// TIA Portal project "Conveyor_LAD_V16_20260903" (V16)

(* hardware
DEVICE "S7-1200 station_1"  S7-1200 Station
   slot 0: "Rack_0"  S7-1200 Rack  Rack  V1.0
   slot 1: "PLC_Conveyor"  CPU 1214C DC/DC/DC  6ES7 214-1AG40-0XB0  V4.4
*)

// ===== PLC "PLC_Conveyor"  CPU 1214C DC/DC/DC =====

VAR_GLOBAL   // PLC tag table "Conveyor_IO_LAD"
   "Conveyor_StartButton" AT %I0.0 : Bool;
   "Conveyor_StopOK" AT %I0.1 : Bool;
   "Conveyor_EStopOK" AT %I0.2 : Bool;
   "Conveyor_OverloadOK" AT %I0.3 : Bool;
   "Conveyor_JamSensor" AT %I0.4 : Bool;
   "Conveyor_ResetButton" AT %I0.5 : Bool;
   "Conveyor_MotorCmd" AT %Q0.0 : Bool;
   "Conveyor_RunLamp" AT %Q0.1 : Bool;
   "Conveyor_FaultLamp" AT %Q0.2 : Bool;
END_VAR

DATA_BLOCK "DB_Conveyor_LAD"   // DB2
{ S7_Optimized_Access := 'TRUE' }
VERSION : 0.1
// stored: InstanceOfName FB_Conveyor_LAD
"FB_Conveyor_LAD"
BEGIN
END_DATA_BLOCK

FUNCTION_BLOCK "FB_Conveyor_LAD"   // FB2, LAD
{ S7_Optimized_Access := 'TRUE' }
   VAR_INPUT
      FirstScan : Bool;
      StartButton : Bool;
      StopOK : Bool;
      EStopOK : Bool;
      OverloadOK : Bool;
      JamSensor : Bool;
      ResetButton : Bool;
      JamTime : Time := T#5s;
   END_VAR
   VAR_OUTPUT
      MotorCmd : Bool;
      RunLamp : Bool;
      FaultLamp : Bool;
   END_VAR
   VAR
      StartPrev : Bool := FALSE;
      RunLatch : Bool := FALSE;
      FaultLatch : Bool := FALSE;
      JamTimer : TON_TIME;
   END_VAR
BEGIN

REGION Network 1: 01 - First scan: reset run latch
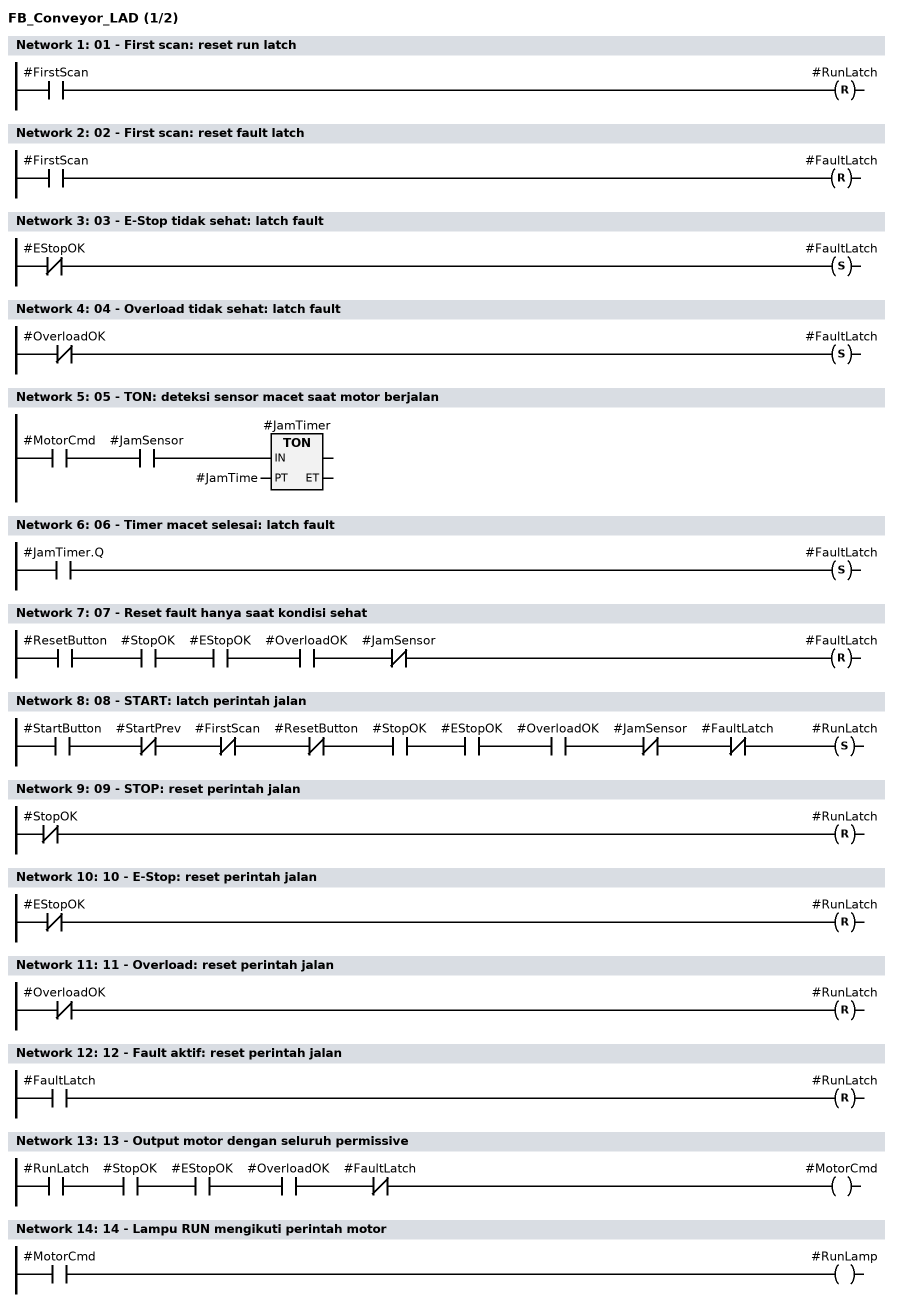
   RUNG wire#powerrail
      Contact( #FirstScan )
      R_Coil( #RunLatch )
   END_RUNG
   // the same network as SCL:
   IF #FirstScan THEN #RunLatch := FALSE; END_IF;
END_REGION

REGION Network 2: 02 - First scan: reset fault latch
   RUNG wire#powerrail
      Contact( #FirstScan )
      R_Coil( #FaultLatch )
   END_RUNG
   // the same network as SCL:
   IF #FirstScan THEN #FaultLatch := FALSE; END_IF;
END_REGION

REGION Network 3: 03 - E-Stop tidak sehat: latch fault
   RUNG wire#powerrail
      I_Contact( #EStopOK )
      S_Coil( #FaultLatch )
   END_RUNG
   // the same network as SCL:
   IF NOT #EStopOK THEN #FaultLatch := TRUE; END_IF;
END_REGION

REGION Network 4: 04 - Overload tidak sehat: latch fault
   RUNG wire#powerrail
      I_Contact( #OverloadOK )
      S_Coil( #FaultLatch )
   END_RUNG
   // the same network as SCL:
   IF NOT #OverloadOK THEN #FaultLatch := TRUE; END_IF;
END_REGION

REGION Network 5: 05 - TON: deteksi sensor macet saat motor berjalan
   #JamTimer(IN := #MotorCmd AND #JamSensor, PT := #JamTime);   // TON
END_REGION

REGION Network 6: 06 - Timer macet selesai: latch fault
   RUNG wire#powerrail
      Contact( #JamTimer.Q )
      S_Coil( #FaultLatch )
   END_RUNG
   // the same network as SCL:
   IF #JamTimer.Q THEN #FaultLatch := TRUE; END_IF;
END_REGION

REGION Network 7: 07 - Reset fault hanya saat kondisi sehat
   RUNG wire#powerrail
      Contact( #ResetButton )
      Contact( #StopOK )
      Contact( #EStopOK )
      Contact( #OverloadOK )
      I_Contact( #JamSensor )
      R_Coil( #FaultLatch )
   END_RUNG
   // the same network as SCL:
   IF #ResetButton AND #StopOK AND #EStopOK AND #OverloadOK AND NOT #JamSensor THEN
       #FaultLatch := FALSE;
   END_IF;
END_REGION

REGION Network 8: 08 - START: latch perintah jalan
   RUNG wire#powerrail
      Contact( #StartButton )
      I_Contact( #StartPrev )
      I_Contact( #FirstScan )
      I_Contact( #ResetButton )
      Contact( #StopOK )
      Contact( #EStopOK )
      Contact( #OverloadOK )
      I_Contact( #JamSensor )
      I_Contact( #FaultLatch )
      S_Coil( #RunLatch )
   END_RUNG
   // the same network as SCL:
   IF #StartButton AND NOT #StartPrev AND NOT #FirstScan AND NOT #ResetButton AND #StopOK AND #EStopOK AND #OverloadOK AND NOT #JamSensor AND NOT #FaultLatch THEN
       #RunLatch := TRUE;
   END_IF;
END_REGION

REGION Network 9: 09 - STOP: reset perintah jalan
   RUNG wire#powerrail
      I_Contact( #StopOK )
      R_Coil( #RunLatch )
   END_RUNG
   // the same network as SCL:
   IF NOT #StopOK THEN #RunLatch := FALSE; END_IF;
END_REGION

REGION Network 10: 10 - E-Stop: reset perintah jalan
   RUNG wire#powerrail
      I_Contact( #EStopOK )
      R_Coil( #RunLatch )
   END_RUNG
   // the same network as SCL:
   IF NOT #EStopOK THEN #RunLatch := FALSE; END_IF;
END_REGION

REGION Network 11: 11 - Overload: reset perintah jalan
   RUNG wire#powerrail
      I_Contact( #OverloadOK )
      R_Coil( #RunLatch )
   END_RUNG
   // the same network as SCL:
   IF NOT #OverloadOK THEN #RunLatch := FALSE; END_IF;
END_REGION

REGION Network 12: 12 - Fault aktif: reset perintah jalan
   RUNG wire#powerrail
      Contact( #FaultLatch )
      R_Coil( #RunLatch )
   END_RUNG
   // the same network as SCL:
   IF #FaultLatch THEN #RunLatch := FALSE; END_IF;
END_REGION

REGION Network 13: 13 - Output motor dengan seluruh permissive
   RUNG wire#powerrail
      Contact( #RunLatch )
      Contact( #StopOK )
      Contact( #EStopOK )
      Contact( #OverloadOK )
      I_Contact( #FaultLatch )
      Coil( #MotorCmd )
   END_RUNG
   // the same network as SCL:
   #MotorCmd := #RunLatch AND #StopOK AND #EStopOK AND #OverloadOK AND NOT #FaultLatch;
END_REGION

REGION Network 14: 14 - Lampu RUN mengikuti perintah motor
   RUNG wire#powerrail
      Contact( #MotorCmd )
      Coil( #RunLamp )
   END_RUNG
   // the same network as SCL:
   #RunLamp := #MotorCmd;
END_REGION

REGION Network 15: 15 - Lampu FAULT mengikuti fault latch
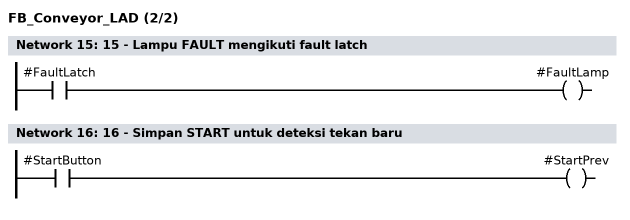
   RUNG wire#powerrail
      Contact( #FaultLatch )
      Coil( #FaultLamp )
   END_RUNG
   // the same network as SCL:
   #FaultLamp := #FaultLatch;
END_REGION

REGION Network 16: 16 - Simpan START untuk deteksi tekan baru
   RUNG wire#powerrail
      Contact( #StartButton )
      Coil( #StartPrev )
   END_RUNG
   // the same network as SCL:
   #StartPrev := #StartButton;
END_REGION
END_FUNCTION_BLOCK

ORGANIZATION_BLOCK "Main"   // OB1, LAD, ProgramCycle
TITLE = "Main Program Sweep (Cycle)"
{ S7_Optimized_Access := 'TRUE' }
VERSION : 0.1
   VAR_INPUT
      Initial_Call : Bool;   // Initial call of this OB
      Remanence : Bool;   // =True, if remanent data are available
   END_VAR
BEGIN

REGION Network 1: Conveyor control - cyclic LAD call
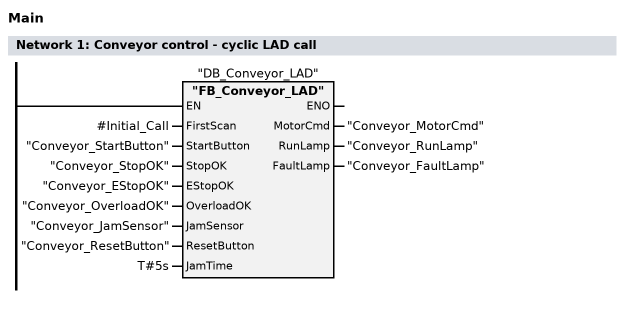
   RUNG wire#powerrail
      "DB_Conveyor_LAD"(FirstScan := #Initial_Call, StartButton := "Conveyor_StartButton", StopOK := "Conveyor_StopOK", EStopOK := "Conveyor_EStopOK", OverloadOK := "Conveyor_OverloadOK", JamSensor := "Conveyor_JamSensor", ResetButton := "Conveyor_ResetButton", JamTime := T#5s, MotorCmd => "Conveyor_MotorCmd", RunLamp => "Conveyor_RunLamp", FaultLamp => "Conveyor_FaultLamp")
   END_RUNG
   // the same network as SCL:
   "DB_Conveyor_LAD"(FirstScan := #Initial_Call,   // "FB_Conveyor_LAD"
                     StartButton := "Conveyor_StartButton",
                     StopOK := "Conveyor_StopOK",
                     EStopOK := "Conveyor_EStopOK",
                     OverloadOK := "Conveyor_OverloadOK",
                     JamSensor := "Conveyor_JamSensor",
                     ResetButton := "Conveyor_ResetButton",
                     JamTime := T#5s,
                     MotorCmd => "Conveyor_MotorCmd",
                     RunLamp => "Conveyor_RunLamp",
                     FaultLamp => "Conveyor_FaultLamp");
END_REGION
END_ORGANIZATION_BLOCK